FUNCTION_BLOCK FB_OmronLD90 EXTENDS FB_ROB_AMR IMPLEMENTS ITF_CommunicationModul
VAR_INPUT
	


	sLoadDeliverReturn: Skill_LoadDeliverReturn;
	sEyes: Skill_ROS2_Eyes;
	ComConfig: ST_CommunicationConfig;
END_VAR
VAR_OUTPUT
  SocketErrorId: UDINT;
END_VAR
VAR
	MissionIndex: INT;
	oldMissionIndex: INT;
	waitTimer: TON;
  fbSocketConnect: FB_SocketConnect;
  fbSocketClose: FB_SocketClose;
  hSocket: T_HSOCKET;
  eConnectionState: eCommunicationState := eCommunicationState.DISCONNECTED;
  _connected: BOOL;
  xConnectRequest: BOOL;
  xDisconnectRequest: BOOL;
  xSocketConnectExecute: BOOL;
  xSocketCloseExecute: BOOL;
  xSocketConnectStarted: BOOL;
  xSocketCloseStarted: BOOL;
END_VAR

CYCLIC_AMR();

ComMachine();

//-------- SKILL SETUP ---------


pA_Skills[1]:=ADR(sLoadDeliverReturn);
pA_Skills[2]:=ADR(sEyes);

sEyes();
sLoadDeliverReturn(Rob:=ADR(THIS^));


//------------------------------------

IF MissionIndex<>oldMissionIndex THEN
	waitTimer(IN:=TRUE, PT:=T#4S);
	oldMissionIndex:=MissionIndex;
END_IF
waitTimer();
IF waitTimer.Q THEN
	waitTimer(IN:=FALSE);
	TargetReached:=TRUE;
	ADSLOGSTR(
    msgCtrlMask := ADSLOG_MSGTYPE_HINT,
    msgFmtStr   := 'Simulated target reached!',
    strArg      := ''
);
	
END_IF

METHOD ComMachine : BOOL
VAR_INPUT
END_VAR
CASE eConnectionState OF


    // =========================================================
    // DISCONNECTED
    // =========================================================

    eCommunicationState.DISCONNECTED:

       _connected := FALSE;


        // Make sure socket handle is cleared
//         hSocket


        // -----------------------------------------------------
        // Connect requested
        // -----------------------------------------------------

        IF xConnectRequest THEN

            xConnectRequest := FALSE;

            // Clear previous errors
            bError := FALSE;
            nErrorId := 0;
            SocketErrorId := 0;

            // Start FB_SocketConnect
            xSocketConnectExecute := TRUE;
            xSocketConnectStarted := TRUE;

            eConnectionState :=
                eCommunicationState.CONNECTING;

        END_IF;


    // =========================================================
    // CONNECTING
    // =========================================================

    eCommunicationState.CONNECTING:

        _connected := FALSE;
        


        // -----------------------------------------------------
        // Execute FB_SocketConnect
        // -----------------------------------------------------

        fbSocketConnect(
            sSrvNetId := '',
            sRemoteHost := ComConfig.sIpAddress,
            nRemotePort := ComConfig.nPort,
            bExecute := xSocketConnectExecute,
            tTimeout := ComConfig.tTimeout
        );


        // Execute must only be TRUE for one cycle
        xSocketConnectExecute := FALSE;


        // -----------------------------------------------------
        // Connection successful
        // -----------------------------------------------------

        IF xSocketConnectStarted
          AND NOT fbSocketConnect.bBusy
            AND NOT fbSocketConnect.bError
//             AND (fbSocketConnect.hSocket <> 0)
        THEN

            hSocket :=
                fbSocketConnect.hSocket;

            _connected := TRUE;
            xSocketConnectStarted := FALSE;
    

            bError := FALSE;
            nErrorId := 0;
            SocketErrorId := 0;

            eConnectionState :=
                eCommunicationState.CONNECTED;

        END_IF;


        // -----------------------------------------------------
        // Connection failed
        // -----------------------------------------------------

        IF NOT fbSocketConnect.bBusy
            AND fbSocketConnect.bError
        THEN

            _connected := FALSE;
          xSocketConnectStarted := FALSE;

            bError := TRUE;

            SocketErrorId :=
                fbSocketConnect.nErrId;

            nErrorId :=
                TO_UINT(fbSocketConnect.nErrId);

//             hSocket := 0;

            eConnectionState :=
                eCommunicationState.ERROR;

        END_IF;


    // =========================================================
    // CONNECTED
    // =========================================================

    eCommunicationState.CONNECTED:

        _connected := TRUE;



        // -----------------------------------------------------
        // Disconnect requested
        // -----------------------------------------------------

        IF xDisconnectRequest THEN

            xDisconnectRequest := FALSE;


            // Start socket close
            xSocketCloseExecute := TRUE;
            xSocketCloseStarted := TRUE;

            eConnectionState :=
                eCommunicationState.DISCONNECTING;

        END_IF;


    // =========================================================
    // DISCONNECTING
    // =========================================================

    eCommunicationState.DISCONNECTING:

        _connected := FALSE;


        // -----------------------------------------------------
        // Execute FB_SocketClose
        // -----------------------------------------------------

        fbSocketClose(
            sSrvNetId := '',
            hSocket := hSocket,
            bExecute := xSocketCloseExecute,
            tTimeout := ComConfig.tTimeout
        );


        // Execute only for one cycle
        xSocketCloseExecute := FALSE;


        // -----------------------------------------------------
        // Socket closed successfully
        // -----------------------------------------------------

        IF xSocketCloseStarted
          AND NOT fbSocketClose.bBusy
            AND NOT fbSocketClose.bError
        THEN

            _connected := FALSE;


            xSocketCloseStarted := FALSE;

            eConnectionState :=
                eCommunicationState.DISCONNECTED;

        END_IF;


        // -----------------------------------------------------
        // Socket close failed
        // -----------------------------------------------------

        IF NOT fbSocketClose.bBusy
            AND fbSocketClose.bError
        THEN

            _connected := FALSE;
          xSocketCloseStarted := FALSE;


            bError := TRUE;

            SocketErrorId :=
                fbSocketClose.nErrId;

            nErrorId :=
                TO_UINT(fbSocketClose.nErrId);

            // The socket should no longer be used
//             hSocket := 0;

            eConnectionState :=
                eCommunicationState.ERROR;

        END_IF;


    // =========================================================
    // ERROR
    // =========================================================

    eCommunicationState.ERROR:

        _connected := FALSE;
        // -----------------------------------------------------
        // Do not attempt to use the socket after an error
        // -----------------------------------------------------

//         hSocket := 0;


        // -----------------------------------------------------
        // A new connection request can recover from the error
        // -----------------------------------------------------

        IF xConnectRequest THEN

            xConnectRequest := FALSE;

            bError := FALSE;
            nErrorId := 0;
            SocketErrorId := 0;

            xSocketConnectExecute := TRUE;
            xSocketConnectStarted := TRUE;

            eConnectionState :=
                eCommunicationState.CONNECTING;

        END_IF;


END_CASE;

CommunicationReady := _connected;
ComMachine := NOT bError;
END_METHOD

{warning 'Add method implementation '}
METHOD Connect : BOOL

Connect := FALSE;

// Already connected
IF eConnectionState = eCommunicationState.CONNECTED THEN
    Connect := TRUE;
    RETURN;
END_IF;

// Already trying to connect
IF eConnectionState = eCommunicationState.CONNECTING THEN
    Connect := TRUE;
    RETURN;
END_IF;

// Don't accept a new connection while disconnecting
IF eConnectionState = eCommunicationState.DISCONNECTING THEN
    RETURN;
END_IF;

// Validate address
IF LEN(ComConfig.sIpAddress) = 0 THEN
    bError := TRUE;
//     ErrorId := 16#1001;
    RETURN;
END_IF;

// Validate port
IF ComConfig.nPort = 0 THEN
    bError := TRUE;
//     ErrorId := 16#1002;
    RETURN;
END_IF;

// Clear previous error
bError := FALSE;
nErrorId := 0;

// Request connection
xConnectRequest := TRUE;

Connect := TRUE;
END_METHOD

{warning 'Add property implementation'}
PROPERTY Connected : BOOL
GET
Connected:=_connected;
END_GET
END_PROPERTY

{warning 'Add method implementation '}
METHOD Disconnect : BOOL
IF eConnectionState = eCommunicationState.DISCONNECTED THEN
      Disconnect := TRUE;
      RETURN;
    END_IF

    xConnectRequest := FALSE;
    xDisconnectRequest := TRUE;
    Disconnect := TRUE;
END_METHOD

METHOD Dock : BOOL
Dock := FALSE;
END_METHOD


  METHOD NavigateToGoal : BOOL
VAR_INPUT
    goal : STRING;
END_VAR
NavigateToGoal := FALSE;

  ADSLOGSTR(
    msgCtrlMask := ADSLOG_MSGTYPE_HINT,
    msgFmtStr   := 'Goes to goal %s',
    strArg      := goal
);

TargetReached:=FALSE;
MissionIndex:=MissionIndex+1;
  NavigateToGoal := TRUE;
END_METHOD

METHOD NavigateToPoint : BOOL
  VAR_INPUT
    point : stPose2D;
  END_VAR
END_METHOD

METHOD PROTECTED OnActivate : eResult
IF bError THEN
    OnActivate := eResult.ERROR;
    ELSIF Connected THEN
      OnActivate := eResult.SUCCESS;
ELSE
      OnActivate := eResult.None;
END_IF
END_METHOD

METHOD PROTECTED OnCleanup : eResult
Disconnect();

    IF eConnectionState <> eCommunicationState.DISCONNECTED THEN
      OnCleanup := eResult.None;
    ELSE
      OnCleanup := eResult.SUCCESS;
    END_IF
END_METHOD

METHOD PROTECTED OnConfigure : eResult
Connect();

    IF bError THEN
      OnConfigure := eResult.ERROR;
    ELSIF Connected THEN
      OnConfigure := eResult.SUCCESS;
    ELSE
      OnConfigure := eResult.None;
    END_IF
END_METHOD

METHOD PROTECTED OnDeactivate : eResult
IF bError THEN
    OnDeactivate := eResult.ERROR;
ELSE
    OnDeactivate := eResult.SUCCESS;
END_IF
END_METHOD

METHOD PROTECTED OnError : eResult
OnError := eResult.SUCCESS;
END_METHOD

METHOD PROTECTED OnShutdown : eResult
Disconnect();

    IF eConnectionState <> eCommunicationState.DISCONNECTED THEN
      OnShutdown := eResult.None;
    ELSIF bError THEN
      OnShutdown := eResult.ERROR;
    ELSE
      OnShutdown := eResult.SUCCESS;
    END_IF
END_METHOD

{warning 'Add method implementation '}
METHOD ResetConnection : BOOL
END_METHOD

METHOD Undock : BOOL
  VAR_INPUT
  END_VAR
END_METHOD

END_FUNCTION_BLOCK

(* stored: Version 1.1.0.1, ProductVersion 3.1.4026.18
   POU FB_OmronLD90: Id {fac74160-c2b3-4f77-bd69-eddf1970c653}, SpecialFunc None
   Folder Communication: Id {2a9c337e-719c-4121-a5a9-4ddfd8584a43}
   Folder MotionControl: Id {94b27a46-e651-4eff-a38f-a2a3d5ee10b5}
   Folder StateControl: Id {67994def-610e-4a0b-a6c8-85df31e22884}
   Method ComMachine: Id {040d86b8-c78e-42d4-a5c1-25c0270b6e14}
   Method Connect: Id {70fa978a-67c6-43be-99fb-d03c8689cf07}
   Property Connected: Id {e71d8962-d52b-46f4-b79d-88e001b39f65}
   Get Get: Id {1724321d-02c7-40cd-942a-414eba41ba06}
   Method Disconnect: Id {c75c2374-9ebb-4dd8-a5bc-f61f0a69c931}
   Method Dock: Id {ed889dfa-89d4-4c82-aa20-11f1706e94ee}
   Method NavigateToGoal: Id {bbbc983d-cf30-4dcf-8a44-55f25ea52986}
   Method NavigateToPoint: Id {d734b238-2cc5-407d-bb20-af9fe27df7a9}
   Method OnActivate: Id {7fa92802-2ede-4193-9973-ad7754d17239}
   Method OnCleanup: Id {7747948a-f8e1-4cdb-8a20-610ab536a0ef}
   Method OnConfigure: Id {c568c508-6321-435c-b7c4-683ad73a8f42}
   Method OnDeactivate: Id {57ce1156-6b80-40b7-8fff-100660e6e779}
   Method OnError: Id {74c0a508-94ea-4785-a0ea-1af2639ff5e5}
   Method OnShutdown: Id {f496723a-9c1c-413c-b4ed-4d78c56c0863}
   Method ResetConnection: Id {1a6fc39d-923f-4cb8-bc55-cd413f8ec29d}
   Method Undock: Id {c887c4e0-0c83-4491-ac2c-d3b9fd05bfa5} *)
